// Implicitly generated code : DO NOT EDIT
FUNCTION CheckDivLReal : LREAL
VAR_INPUT
    divisor:LREAL;
END_VAR

// Implicitly generated code : Only an Implementation suggestion
{noflow}
IF divisor = 0 THEN
    CheckDivLReal:=1;
ELSE
    CheckDivLReal:=divisor;
END_IF;
{flow}

END_FUNCTION

(* stored: Version 1.1.0.1
   POU CheckDivLReal: Id {4afc626f-14dd-4b1a-a5dd-77cfb7d31d43}, SpecialFunc CheckDivReal64 *)
